FUNCTION_BLOCK OneIsolator_Latch
VAR_INPUT
	ISO_Status: BOOL;
	OA_IsoReset: BOOL;
END_VAR
VAR_OUTPUT
	ISO_Fault: BOOL;
END_VAR
VAR
END_VAR

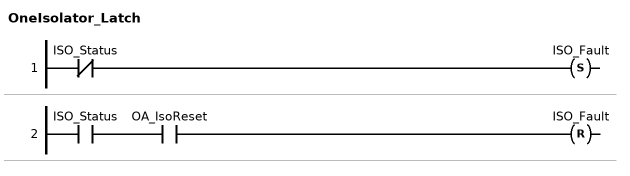
// NETWORK 1
ISO_Fault S= NOT ISO_Status;

// NETWORK 2
ISO_Fault R= ISO_Status AND OA_IsoReset;

END_FUNCTION_BLOCK

(* stored: Version 1.1.0.1, ProductVersion 3.1.4024.12
   POU OneIsolator_Latch: Id {26952cf3-0ef3-4675-9e74-f29f08225849}, SpecialFunc None *)
